# B&R Automation Studio project lab1
Automation Studio 4.5.2.102

## Configuration labBR

### Task classes (Cpu.sw)
```
Cyclic#4:
  Program <- Program.prg
Libraries: MotorCtrl
```

## Logical view

### Program Logical/Program (ANSIC)

#### Variables.var
```iecst
VAR
	fb_motor3 : FB_Motor;
	fb_motor2 : FB_Motor;
	fb_controller : FB_Regulator;
	fb_motor : FB_Motor;
	speed : REAL;
	Enable : BOOL;
	count : REAL;
	integrator : FB_Integrator;
	fb_controller2 : FB_Regulator;
END_VAR
```

#### Cyclic.c
```c
#include <bur/plctypes.h>

#ifdef _DEFAULT_INCLUDES
	#include <AsDefault.h>
#endif

void _CYCLIC ProgramCyclic(void)
{
	if(Enable ==1)
	{
		count+=10;
		if (count >=400 && count <=2000) speed = 40;
		else {
			speed = 5;
		}
		if(count >= 2000){
			count = 0;
		}
	}
	else speed = 0;

	fb_controller.e = speed-fb_motor.w;
	fb_controller2.e = speed-fb_motor3.w;

	fb_motor2.u = speed*fb_motor2.ke;
	fb_motor.u = fb_controller.u*fb_motor.ke;
	fb_motor3.u = fb_controller2.u*fb_motor3.ke;

	FB_Regulator(&fb_controller);
	FB_Regulator(&fb_controller2);
	FB_Motor(&fb_motor);
	FB_Motor(&fb_motor2);
	FB_Motor(&fb_motor3);
}
```

#### Init.c
```c
#include <bur/plctypes.h>

#ifdef _DEFAULT_INCLUDES
	#include <AsDefault.h>
#endif

void _INIT ProgramInit(void)
{
	Enable = 1;
	count = 0;
	speed = 0;

	fb_motor.dt = 0.01;
	fb_motor.ke = 0.24;
	fb_motor.Tm = 0.1;

	fb_motor2.dt = 0.01;
	fb_motor2.ke = 0.24;
	fb_motor2.Tm = 0.1;

	fb_motor3.dt = 0.01;
	fb_motor3.ke = 0.24;
	fb_motor3.Tm = 0.1;

	fb_controller.dt = 0.01;
	fb_controller.k_p = 5;
	fb_controller.k_i = 6;

	fb_controller2.dt = 0.01;
	fb_controller2.k_p = 0.24*3;
	fb_controller2.k_i = 7.2;

	fb_controller.max_abs_value = 24;
}
```

### Package Logical/Libraries - Global libraries

### Library Logical/Libraries/MotorCtrl

#### MotorCtrl.fun
```iecst
{REDUND_ERROR} FUNCTION_BLOCK FB_Motor (*TODO: Add your comment here*) (*$GROUP=User,$CAT=User,$GROUPICON=User.png,$CATICON=User.png*)
	VAR_INPUT
		u : REAL;
	END_VAR
	VAR_OUTPUT
		w : REAL;
		phi : REAL;
	END_VAR
	VAR
		integrator : FB_Integrator;
		Tm : REAL;
		ke : REAL;
		dt : REAL;
	END_VAR
END_FUNCTION_BLOCK

{REDUND_ERROR} FUNCTION_BLOCK FB_Integrator (*TODO: Add your comment here*) (*$GROUP=User,$CAT=User,$GROUPICON=User.png,$CATICON=User.png*)
	VAR_INPUT
		in : REAL;
	END_VAR
	VAR_OUTPUT
		out : REAL;
	END_VAR
	VAR
		dt : REAL;
	END_VAR
END_FUNCTION_BLOCK

{REDUND_ERROR} FUNCTION_BLOCK FB_Regulator (*TODO: Add your comment here*) (*$GROUP=User,$CAT=User,$GROUPICON=User.png,$CATICON=User.png*)
	VAR_INPUT
		e : REAL;
	END_VAR
	VAR_OUTPUT
		u : REAL;
	END_VAR
	VAR
		k_p : REAL;
		k_i : REAL;
		integrator : FB_Integrator;
		iyOld : REAL;
		max_abs_value : REAL;
		dt : REAL;
		e_p : REAL;
	END_VAR
END_FUNCTION_BLOCK
```

#### FB_Integrator.c
```c
#include <bur/plctypes.h>
#ifdef __cplusplus
	extern "C"
	{
#endif
	#include "MotorCtrl.h"
#ifdef __cplusplus
	};
#endif
/* TODO: Add your comment here */
void FB_Integrator(struct FB_Integrator* inst)
{
	inst->out+=inst->in;
}
```

#### FB_Motor.c
```c
#include <bur/plctypes.h>
#ifdef __cplusplus
	extern "C"
	{
#endif
	#include "MotorCtrl.h"
#ifdef __cplusplus
	};
#endif
/* TODO: Add your comment here */
void FB_Motor(struct FB_Motor* inst)
{
	inst->integrator.in = (inst->u*(1/inst->ke)-inst->w)*(inst->dt/inst->Tm);
	FB_Integrator(&(inst->integrator));

	inst->w = inst->integrator.out;
	inst->integrator.in=inst->w*inst->dt;
	FB_Integrator(&(inst->integrator));

	inst->phi=inst->integrator.out;
}
```

#### FB_Regulator.c
```c
#include <bur/plctypes.h>
#ifdef __cplusplus
	extern "C"
	{
#endif
	#include "MotorCtrl.h"
#ifdef __cplusplus
	};
#endif
/* TODO: Add your comment here */
void FB_Regulator(struct FB_Regulator* inst)
{
	/*TODO: Add your code here*/
	inst->integrator.in = inst->e*inst->k_i*inst->dt + inst->iyOld;
	FB_Integrator(&(inst->integrator));

	inst->e_p = inst->e*inst->k_p;

	if (inst->e_p< inst->max_abs_value||inst->e_p > -inst->max_abs_value);
		else
	{
		if (inst->e_p > 0) inst->e_p = inst->max_abs_value;
		else inst->e_p = -inst->max_abs_value;
	}

	inst->e_p += inst->integrator.out;
	if (inst->e_p< inst->max_abs_value||inst->e_p> -inst->max_abs_value) inst ->u = inst->e_p;

	else
	{
		if (inst->e_p > 0) inst ->u = inst->max_abs_value;
		else inst ->u = -inst ->max_abs_value;
	}

	inst->iyOld = inst ->u - inst->e_p;
}
```

Listed in the project but not available here: Logical/Global.typ, Logical/Global.var
